DATA_BLOCK "DB_BSO_Type"
TITLE =%version: 0.10 % CN: 20
//History:
//This version  %created_by: nlhdl %
//              %date_created: Thursday, January 25, 2018 8:36:22 AM %
//              %release: VI_GEN/RA_Dev %
//
//Modification History:                                   By:    Date:     Rev:
//----------------------------------------------------  -------  --------  -----
//ra#27505: Add unexpected data WN and ER to status     nlHdL    25-01-18   0.10
//ra#26202: Error text Invalid Barcode                  nlHdL    27-11-17   0.09
//ra#24858: BSO add warnings to type DB                 nlHdL    03-10-17   0.08
//ra#16735: DI NON_RETAIN PLC Memory                    nlHdL    13-12-16   0.07
//ra#15851: Add BSO from RAW to General Library         nlHdL    19-07-16   0.06
//ra#15851: Add BSO from RAW to General Library         nlHdL    19-07-16   0.06
//7324: ECS-P General from the RD to RA for platform    nlHdL    06-07-15   0.06
//15797: Keyword release added                          nlwwij   26-09-13   0.06
//CR5856 Changed ATR into BSO                           nlJBax   26-10-10   0.05
//CR5737 Removed warning message details                inpna    04-10-10   0.04
//CR5712 Not used errors have number -1                 nlHdL    24-09-10   0.03
//Added the Text number                                 inpna    23-09-10   0.02
//Initial Revision                                      inpna    17-09-10   0.01
//
FAMILY : General
VERSION : 0.0
NON_RETAIN


  STRUCT
   Type_Component : BYTE ;	//Type of the component (1 = Section, 0 = Other)
   Record_Length : BYTE  := B#16#16;	//Number of the Detailed Status in the UDT
   Status : ARRAY  [1 .. 16 ] OF "UDT_Comp_Status";
  END_STRUCT ;
BEGIN
   Type_Component := B#16#0;
   Record_Length := B#16#16;
   Status[1].HMI_Text_Number := 48;
   Status[1].Overall_Status_Relation := B#16#5;
   Status[1].General_Status_Relation := B#16#4;
   Status[2].HMI_Text_Number := 49;
   Status[2].Overall_Status_Relation := B#16#4;
   Status[2].General_Status_Relation := B#16#3;
   Status[3].HMI_Text_Number := -1;
   Status[3].Overall_Status_Relation := B#16#0;
   Status[3].General_Status_Relation := B#16#0;
   Status[4].HMI_Text_Number := -1;
   Status[4].Overall_Status_Relation := B#16#0;
   Status[4].General_Status_Relation := B#16#0;
   Status[5].HMI_Text_Number := 73;
   Status[5].Overall_Status_Relation := B#16#5;
   Status[5].General_Status_Relation := B#16#4;
   Status[6].HMI_Text_Number := 72;
   Status[6].Overall_Status_Relation := B#16#5;
   Status[6].General_Status_Relation := B#16#4;
   Status[7].HMI_Text_Number := 60;
   Status[7].Overall_Status_Relation := B#16#4;
   Status[7].General_Status_Relation := B#16#3;
   Status[8].HMI_Text_Number := 61;
   Status[8].Overall_Status_Relation := B#16#4;
   Status[8].General_Status_Relation := B#16#3;
   Status[9].HMI_Text_Number := 56;
   Status[9].Overall_Status_Relation := B#16#4;
   Status[9].General_Status_Relation := B#16#3;
   Status[10].HMI_Text_Number := 67;
   Status[10].Overall_Status_Relation := B#16#4;
   Status[10].General_Status_Relation := B#16#3;
   Status[11].HMI_Text_Number := 66;
   Status[11].Overall_Status_Relation := B#16#4;
   Status[11].General_Status_Relation := B#16#3;
   Status[12].HMI_Text_Number := 55;
   Status[12].Overall_Status_Relation := B#16#4;
   Status[12].General_Status_Relation := B#16#3;
   Status[13].HMI_Text_Number := 51;
   Status[13].Overall_Status_Relation := B#16#4;
   Status[13].General_Status_Relation := B#16#3;
   Status[14].HMI_Text_Number := 53;
   Status[14].Overall_Status_Relation := B#16#4;
   Status[14].General_Status_Relation := B#16#3;
   Status[15].HMI_Text_Number := -1;
   Status[15].Overall_Status_Relation := B#16#0;
   Status[15].General_Status_Relation := B#16#0;
   Status[16].HMI_Text_Number := -1;
   Status[16].Overall_Status_Relation := B#16#0;
   Status[16].General_Status_Relation := B#16#0;
END_DATA_BLOCK

